# EPICS substitutions: apps/CaenHVApp/db/CaenHV_crate4.substitutions
file "db/AS503_Chan.template" {
pattern
    {P,      H,  S,   V}
    {hchv,   4,  00,  000}
    {hchv,   4,  00,  001}
    {hchv,   4,  00,  002}
    {hchv,   4,  00,  003}
    {hchv,   4,  00,  004}
    {hchv,   4,  00,  005}
    {hchv,   4,  00,  006}
    {hchv,   4,  00,  007}
    {hchv,   4,  00,  008}
    {hchv,   4,  00,  009}
    {hchv,   4,  00,  010}
    {hchv,   4,  00,  011}
    {hchv,   4,  00,  012}
    {hchv,   4,  00,  013}
    {hchv,   4,  00,  014}
    {hchv,   4,  00,  015}
}
file "db/AS503_Chan.template" {
pattern
    {P,      H,  S,   V}
    {hchv,   4,  01, 000}
    {hchv,   4,  01, 001}
    {hchv,   4,  01, 002}
    {hchv,   4,  01, 003}
    {hchv,   4,  01, 004}
    {hchv,   4,  01, 005}
    {hchv,   4,  01, 006}
    {hchv,   4,  01, 007}
    {hchv,   4,  01, 008}
    {hchv,   4,  01, 009}
    {hchv,   4,  01, 010}
    {hchv,   4,  01, 011}
    {hchv,   4,  01, 012}
    {hchv,   4,  01, 013}
    {hchv,   4,  01, 014}
    {hchv,   4,  01, 015}
}
file "db/AS503_Chan.template" {
pattern
    {P,      H,  S,   V}
    {hchv,   4,  02, 000}
    {hchv,   4,  02, 001}
    {hchv,   4,  02, 002}
    {hchv,   4,  02, 003}
    {hchv,   4,  02, 004}
    {hchv,   4,  02, 005}
    {hchv,   4,  02, 006}
    {hchv,   4,  02, 007}
    {hchv,   4,  02, 008}
    {hchv,   4,  02, 009}
    {hchv,   4,  02, 010}
    {hchv,   4,  02, 011}
    {hchv,   4,  02, 012}
    {hchv,   4,  02, 013}
    {hchv,   4,  02, 014}
    {hchv,   4,  02, 015}
}
file "db/AS503_Chan.template" {
pattern
    {P,      H,  S,   V}
    {hchv,   4,  03, 000}
    {hchv,   4,  03, 001}
    {hchv,   4,  03, 002}
    {hchv,   4,  03, 003}
    {hchv,   4,  03, 004}
    {hchv,   4,  03, 005}
    {hchv,   4,  03, 006}
    {hchv,   4,  03, 007}
    {hchv,   4,  03, 008}
    {hchv,   4,  03, 009}
    {hchv,   4,  03, 010}
    {hchv,   4,  03, 011}
    {hchv,   4,  03, 012}
    {hchv,   4,  03, 013}
    {hchv,   4,  03, 014}
    {hchv,   4,  03, 015}
}
